INTERFACE I_VarStringBuffer EXTENDS I_VarByteBufferBase

METHOD Push : BOOL
VAR_INPUT
	sInputString	: REFERENCE TO T_MaxString;
END_VAR
END_METHOD

END_INTERFACE

(* stored: Version 1.1.0.1
   Itf I_VarStringBuffer: Id {88388f11-4090-4f89-8c54-777e8983e069}
   Method Push: Id {3e12aae4-b3d2-46ea-bf2c-f63cb44f3cbe} *)
